FUNCTION_BLOCK logiBUS_AI_IDA (* Composite FB for analog double word input data *)
  (* Standard: 61499-2; Description: Copyright (c) 2026 HR Agrartechnik GmbH This program and the accompanying materials are made available under the terms of the Eclipse Public License 2.0 which is available at https://www.eclipse.org/legal/epl-2.0/ SPDX-License-Identifier: EPL-2.0 if AnalogInput_hysteresis = 0, then TimeDelta cannot be 0. set TimeDelta to 16#FFFFFFFF to deactivate cyclic processing, and onyl indicate Changes in Value. *)
  (* Version 1.0, 2026-02-23, Franz Höpfinger, HR Agrartechnik GmbH *)
  PACKAGE logiBUS::io::AI;
  IMPORT logiBUS::io::AI::logiBUS_AI::Invalid;
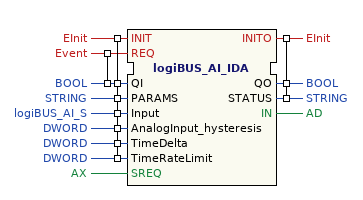
  EVENT_INPUT
    INIT : EInit WITH QI, PARAMS, Input, AnalogInput_hysteresis, TimeDelta, TimeRateLimit; (* Service Initialization *)
    REQ WITH QI; (* Service Request *)
  END_EVENT
  EVENT_OUTPUT
    INITO : EInit WITH QO, STATUS; (* Initialization Confirm *)
  END_EVENT
  VAR_INPUT
    QI : BOOL; (* Event Input Qualifier *)
    PARAMS : STRING; (* Service Parameters *)
    Input : logiBUS::io::AI::logiBUS_AI_S := Invalid; (* Identify the Input Input_I1..I8 *)
    AnalogInput_hysteresis : DWORD;
    TimeDelta : DWORD := 250; (* After How many ms an IND *)
    TimeRateLimit : DWORD := 100; (* Maximum 1 IND in how many ms. (< delta) *)
  END_VAR
  VAR_OUTPUT
    QO : BOOL; (* Event Output Qualifier *)
    STATUS : STRING; (* Service Status *)
  END_VAR
  SOCKETS
    SREQ : adapter::types::unidirectional::AX; (* Service Request *)
  END_SOCKETS
  PLUGS
    IN : adapter::types::unidirectional::AD; (* Input data from resource *)
  END_PLUGS
  FBS
    AI : logiBUS::io::AI::logiBUS_AI_ID;
    E_R_TRIG : iec61499::events::E_R_TRIG;
  END_FBS
  EVENT_CONNECTIONS
    INIT TO AI.INIT;
    AI.INITO TO INITO;
    AI.IND TO IN.E1;
    AI.CNF TO IN.E1;
    REQ TO AI.REQ;
    E_R_TRIG.EO TO AI.REQ;
    SREQ.E1 TO E_R_TRIG.EI;
  END_CONNECTIONS
  DATA_CONNECTIONS
    AI.IN TO IN.D1;
    QI TO AI.QI;
    PARAMS TO AI.PARAMS;
    AI.QO TO QO;
    AI.STATUS TO STATUS;
    Input TO AI.Input;
    AnalogInput_hysteresis TO AI.AnalogInput_hysteresis;
    SREQ.D1 TO E_R_TRIG.QI;
    TimeDelta TO AI.TimeDelta;
    TimeRateLimit TO AI.TimeRateLimit;
  END_CONNECTIONS
END_FUNCTION_BLOCK
